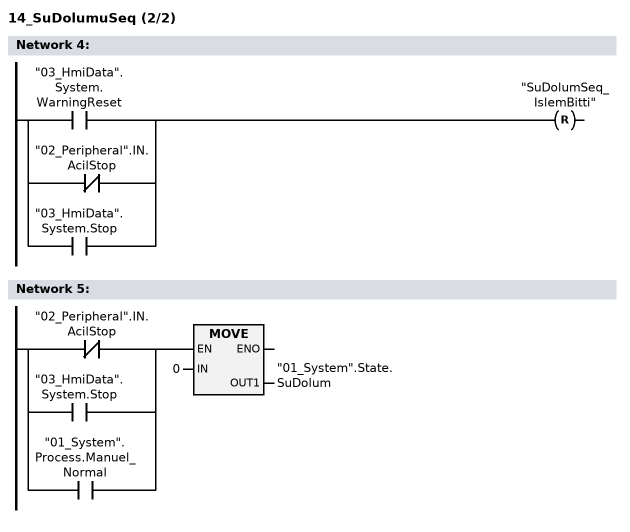
   RUNG wire#powerrail
      Contact( "03_HmiData".System.WarningReset )
      wire#w1
      R_Coil( "SuDolumSeq_IslemBitti" )
   END_RUNG
   RUNG wire#powerrail
      I_Contact( "02_Peripheral".IN.AcilStop )
   END_RUNG wire#w1
   RUNG wire#powerrail
      Contact( "03_HmiData".System.Stop )
   END_RUNG wire#w1
   // the same network as SCL:
   IF "03_HmiData".System.WarningReset OR NOT "02_Peripheral".IN.AcilStop OR "03_HmiData".System.Stop THEN
       "SuDolumSeq_IslemBitti" := FALSE;
   END_IF;
END_REGION

REGION Network 5
   RUNG wire#powerrail
      I_Contact( "02_Peripheral".IN.AcilStop )
      wire#w1
      Move(in := 0, out1 => "01_System".State.SuDolum)
   END_RUNG
   RUNG wire#powerrail
      Contact( "03_HmiData".System.Stop )
   END_RUNG wire#w1
   RUNG wire#powerrail
      Contact( "01_System".Process.Manuel_Normal )
   END_RUNG wire#w1
   // the same network as SCL:
   IF NOT "02_Peripheral".IN.AcilStop OR "03_HmiData".System.Stop OR "01_System".Process.Manuel_Normal THEN
       "01_System".State.SuDolum := 0;
   END_IF;
END_REGION
END_FUNCTION

ORGANIZATION_BLOCK "Main"   // OB1, FBD, ProgramCycle
TITLE = "Main Program Sweep (Cycle)"
{ S7_Optimized_Access := 'TRUE' }
VERSION : 0.1
   VAR_INPUT
      Initial_Call : Bool;   // Initial call of this OB
      Remanence : Bool;   // =True, if remanent data are available
   END_VAR
BEGIN

REGION Network 1: Manuel
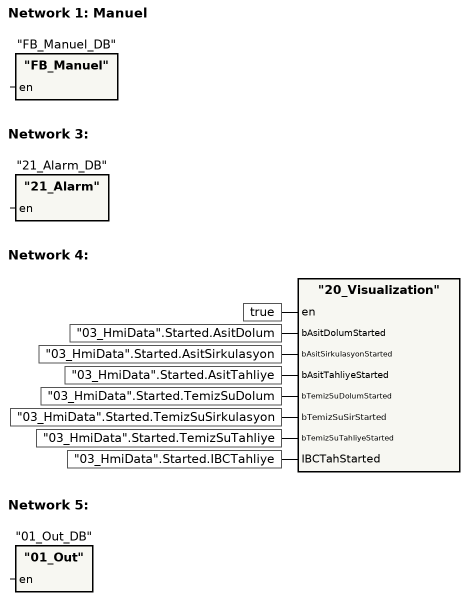
   "FB_Manuel_DB"();   // "FB_Manuel"
END_REGION

REGION Network 2 (SCL): Otomatik sekanslar
   "11_AsitDolumSeq"();
   "12_AsitSirkulasyonSeq"();
   "13_AsitTahliyeSeq"();
   "14_SuDolumuSeq"();
   "15_SuSirkulasyonSeq"();
   "16_SuTahliyeSeq"();
   "17_IBCTahliyeSeq"();

   "22_Peripheral"();
   "23_UyariLambalari"();

   "Always_On" := true;
END_REGION

REGION Network 3
   "21_Alarm_DB"();   // "21_Alarm"
END_REGION

REGION Network 4
   IF true THEN
       "20_Visualization"(bAsitDolumStarted := "03_HmiData".Started.AsitDolum,
                          bAsitSirkulasyonStarted := "03_HmiData".Started.AsitSirkulasyon,
                          bAsitTahliyeStarted := "03_HmiData".Started.AsitTahliye,
                          bTemizSuDolumStarted := "03_HmiData".Started.TemizSuDolum,
                          bTemizSuSirStarted := "03_HmiData".Started.TemizSuSirkulasyon,
                          bTemizSuTahliyeStarted := "03_HmiData".Started.TemizSuTahliye,
                          IBCTahStarted := "03_HmiData".Started.IBCTahliye);
   END_IF;
END_REGION

REGION Network 5
   "01_Out_DB"();   // "01_Out"
END_REGION
END_ORGANIZATION_BLOCK

ORGANIZATION_BLOCK "Time error interrupt"   // OB80, LAD, TimeErrorInterrupt
{ S7_Optimized_Access := 'TRUE' }
VERSION : 0.1
   VAR_INPUT
      Fault_ID : Byte;   // Fault identifier
      Csg_OBnr : OB_Any;   // Number of OB causing the error
      Csg_Prio : UInt;   // Priority of OB causing the error
   END_VAR
BEGIN
END_ORGANIZATION_BLOCK

ORGANIZATION_BLOCK "Pull or plug of modules"   // OB83, LAD, PullPlug
{ S7_Optimized_Access := 'TRUE' }
VERSION : 0.1
   VAR_INPUT
      LADDR : Hw_Io;   // Hardware identifier
      Event_Class : Byte;   // 16#38/39: module inserted, removed
      Fault_ID : Byte;   // Fault identifier
   END_VAR
BEGIN
END_ORGANIZATION_BLOCK

ORGANIZATION_BLOCK "Rack or station failure"   // OB86, LAD, RackStationFailure
{ S7_Optimized_Access := 'TRUE' }
VERSION : 0.1
   VAR_INPUT
      LADDR : Hw_Device;   // Hardware identifier
      Event_Class : Byte;   // Event class
      Fault_ID : Byte;   // Fault identifier
   END_VAR
BEGIN
END_ORGANIZATION_BLOCK

ORGANIZATION_BLOCK "Startup"   // OB100, LAD, Startup
TITLE = "Complete Restart"
{ S7_Optimized_Access := 'TRUE' }
VERSION : 0.1
   VAR_INPUT
      LostRetentive : Bool;   // True if retentive data are lost
      LostRTC : Bool;   // True if date and time are lost
   END_VAR
BEGIN

REGION Network 1
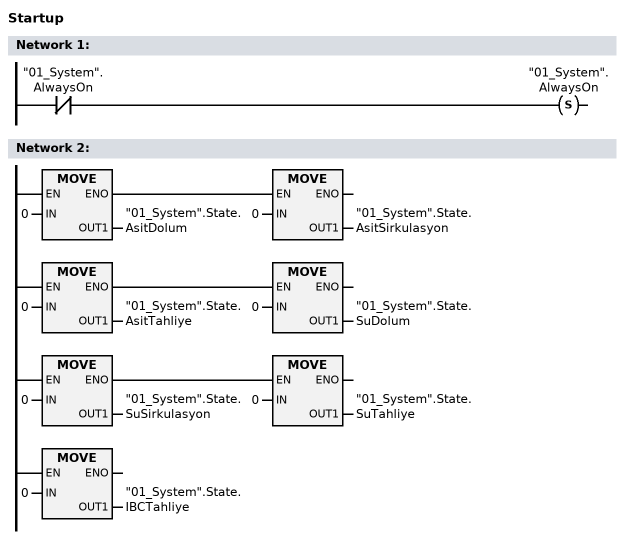
   RUNG wire#powerrail
      I_Contact( "01_System".AlwaysOn )
      S_Coil( "01_System".AlwaysOn )
   END_RUNG
   // the same network as SCL:
   IF NOT "01_System".AlwaysOn THEN "01_System".AlwaysOn := TRUE; END_IF;
END_REGION

REGION Network 2
   RUNG wire#powerrail
      Move(in := 0, out1 => "01_System".State.AsitDolum)
      Move(in := 0, out1 => "01_System".State.AsitSirkulasyon)
   END_RUNG
   RUNG wire#powerrail
      Move(in := 0, out1 => "01_System".State.AsitTahliye)
      Move(in := 0, out1 => "01_System".State.SuDolum)
   END_RUNG
   RUNG wire#powerrail
      Move(in := 0, out1 => "01_System".State.SuSirkulasyon)
      Move(in := 0, out1 => "01_System".State.SuTahliye)
   END_RUNG
   RUNG wire#powerrail
      Move(in := 0, out1 => "01_System".State.IBCTahliye)
   END_RUNG
   // the same network as SCL:
   "01_System".State.AsitDolum := 0;
   "01_System".State.AsitSirkulasyon := 0;
   "01_System".State.AsitTahliye := 0;
   "01_System".State.SuDolum := 0;
   "01_System".State.SuSirkulasyon := 0;
   "01_System".State.SuTahliye := 0;
   "01_System".State.IBCTahliye := 0;
END_REGION
END_ORGANIZATION_BLOCK